TYPE ST_SystemIO :
STRUCT
	
	DI_EL1809 		: ST_EL1809; 
    DO_EL2809 		: ST_EL2809; 
    AI_EL3058 		: ST_EL3058; 

END_STRUCT
END_TYPE

(* stored: Version 1.1.0.1, ProductVersion 3.1.4024.15
   DUT ST_SystemIO: Id {e9a42a03-e182-4cc0-ba21-cd10f789db51} *)
